FUNCTION_BLOCK FB_AlarmMAIN(*报警主功能块,请调用一次*)
VAR_INPUT
END_VAR
VAR_OUTPUT
	EventId:			DINT;(*报警号.有报警时会轮询输出有报警的id号*)
   	EventMessage:       WSTRING(255);(*报警信息.有报警时会轮询输出有报警的id信息*)
	EventAlive:			BOOL;(*当前有报警*)
	EventClass:			Alm_EventClass;(*当前的最大报警等级*)
  	NoStopAlarm:        BOOL;(*有小于7的报警,不停机报警*)
   	StopAlarm:          BOOL;(*有大于6的报警,停机报警*)
   	ShowlampOn:         BOOL;(*报警灯亮*)
   	FalshLamp:          BOOL;(*报警灯闪亮.有报警时该信号闪烁输出*)

	AutoRunOff:			BOOL;(*退出自动循环*)
	AlarmAction1:		BOOL;(*用户定义报警动作*)(*例如定义为黄灯亮,则有报警号有触发时,该输出信号为1*)
	AlarmAction2:		BOOL;(*用户定义报警动作*)
	AlarmAction3:		BOOL;(*用户定义报警动作*)
	AlarmAction4:		BOOL;(*用户定义报警动作*)
	AlarmAction5:		BOOL;(*用户定义报警动作*)
	AlarmAction6:		BOOL;(*用户定义报警动作*)
	AlarmAction7:		BOOL;(*用户定义报警动作*)
	AlarmAction8:		BOOL;(*用户定义报警动作*)
END_VAR
VAR
	nConut:                          DINT;
   	fbFreePluse:                     TON;
	m:                               DINT;
	Resul:                           DINT;
	n:                               DINT;
	R_TRIG_AlarmShow:        		 R_TRIG;
	R_TRIG_AlarmAlive:          	 R_TRIG;
	FB_FreePluse_AlarmShow: 		 TON;
	FB_FreePluse_AlarmAlive: 		 TON;
	F_TRIG_bHMIClearHistory: 		 F_TRIG;
	F_TRIG_EventAlive: 				 F_TRIG;
	InstLocalSystemTime:			 FB_LocalSystemTime;
END_VAR

(*Set Signal*)
 	EventAlive:=ShowlampOn:=AlarmAction1:=AlarmAction2:=AlarmAction3:=FALSE;
  	AlarmAction4:=AlarmAction5:=AlarmAction6:=AlarmAction7:=AlarmAction8:=FALSE;
	AutoRunOff :=	FALSE;(*退出自动循环*)
   	EventClass :=	0;

FOR nConut :=cnAlarmFirst TO cnAlarmLast DO
	    EventAlive :=	EventAlive OR AlarmActionArray[nConut].EventAlive;
	    ShowlampOn :=	ShowlampOn OR AlarmActionArray[nConut].ShowlampOn;
	    AlarmAction1:=	AlarmAction1 OR AlarmActionArray[nConut].AlarmAction1;
	    AlarmAction2:=	AlarmAction2 OR AlarmActionArray[nConut].AlarmAction2;
	    AlarmAction3:=	AlarmAction3 OR AlarmActionArray[nConut].AlarmAction3;
	    AlarmAction4:=	AlarmAction4 OR AlarmActionArray[nConut].AlarmAction4;
	    AlarmAction5:=	AlarmAction5 OR AlarmActionArray[nConut].AlarmAction5;
	    AlarmAction6:=	AlarmAction6 OR AlarmActionArray[nConut].AlarmAction6;
	    AlarmAction7:=	AlarmAction7 OR AlarmActionArray[nConut].AlarmAction7;
	    AlarmAction8:=	AlarmAction8 OR AlarmActionArray[nConut].AlarmAction8;
	    AutoRunOff :=	AutoRunOff 	OR AlarmActionArray[nConut].AutoRunOff;
	    EventClass  :=	MAX(EventClass,AlarmActionArray[nConut].EventClass);
END_FOR

(*Flash lamp*)
R_TRIG_AlarmShow(CLK:=ShowlampOn  );
IF ShowlampOn THEN              (****有报警时，先初始化时间输入为FALSE，灯亮，然后开始下步TON运行1S，闪灯状态变化
                                      优点：一有报警，就灯亮，避免有报警时过1S灯才亮*)
	IF R_TRIG_AlarmShow.Q THEN
		fbFreePluse(IN:=FALSE);
		FalshLamp:=TRUE;
	END_IF
	fbFreePluse(IN:=NOT fbFreePluse.Q,PT:=T#1S);
	IF fbFreePluse.Q THEN
		FalshLamp:=NOT FalshLamp;
	END_IF
ELSE
	FalshLamp:=FALSE;
END_IF



(*Action*)
AlarmAlive();
AlarmHMI();
AlarmShow();

(*Set Action*)
IF EventAlive THEN
     IF EventClass>6 THEN
         StopAlarm:=TRUE;
         NoStopAlarm:=FALSE;
     ELSE
         StopAlarm:=FALSE;
         NoStopAlarm:=TRUE;
    END_IF
ELSE
    StopAlarm:=FALSE;
    NoStopAlarm:=FALSE;
    EventId:=0;
    EventMessage:="";
    Alm_iHMIAlarmID:=0;
END_IF

	//获取系统时间
	InstLocalSystemTime(
		sNetID		:= '',
		bEnable		:= TRUE,
		dwCycle		:= 1,
		systemTime	=> tActSystemTime,
		);

ACTION AlarmAlive:
(*总报警数有n个，用其中有报警的[2],[4]赋值给激活报警m[1],[2],m自加1，然后循环比较m-20,把信息格式化*)
(*-----------------------------------当前报警列表显示-----------------------------*)
R_TRIG_AlarmAlive(CLK:=EventAlive);
IF EventAlive THEN
	IF R_TRIG_AlarmAlive.Q THEN
   	 	FB_FreePluse_AlarmAlive(In:=FALSE);
	END_IF
    FB_FreePluse_AlarmAlive(In:= NOT FB_FreePluse_AlarmAlive.Q,PT:=T#1S );
    IF FB_FreePluse_AlarmAlive.Q OR R_TRIG_AlarmAlive.Q THEN
         n:=cnAlarmFirst;
         m:=cnAlmActiveFirst;
          FOR n:=cnAlarmFirst TO cnAlarmLast DO     (*把所有报警赋值到当前激活报警数组*)
               IF AlarmActionArray[n].EventAlive THEN
                    AlarmActiveArray[m].EventId       :=AlarmActionArray[n].EventId;
                   	AlarmActiveArray[m].EventMessage  :=AlarmActionArray[n].EventMessage;						
                    AlarmActiveArray[m].EventTime     :=AlarmActionArray[n].EventTime;
                  	m:=m+1;
                    IF m>cnAlmActiveLast THEN
                       n:=32766;  (*exit FOR*)
                    END_IF
               END_IF
         END_FOR
         IF m<cnAlmActiveLast THEN
               FOR n:=m TO cnAlmActiveLast DO
                   AlarmActiveArray[n].EventId:=0;
                 	AlarmActiveArray[n].EventMessage:="";
                   	AlarmActiveArray[n].EventTime:=DT#2000-01-01-00:00;
             END_FOR
          END_IF
    END_IF
END_IF
(*当报警消失时,把显示列表内容清空*)
F_TRIG_EventAlive(CLK:=EventAlive );
IF F_TRIG_EventAlive.Q THEN
	FOR n:=cnAlmActiveFirst TO cnAlmActiveLast DO 
		AlarmActiveArray[n].EventId:=0;
		AlarmActiveArray[n].EventMessage:="";
		AlarmActiveArray[n].EventTime:=DT#2016-01-01-00:00;
	END_FOR
END_IF
END_ACTION

ACTION AlarmHMI:


(*``````````````````````````````````````````清除历史报警`````````````````````````````````````*)
F_TRIG_bHMIClearHistory(CLK:=Alm_bHMIClearHistory  );
IF F_TRIG_bHMIClearHistory.Q THEN
       FOR n:=cnAlmHistoryFirst TO cnAlmHistoryLast DO
             AlarmHistoryArray[n].EventId:=0;
             AlarmHistoryArray[n].EventMessage:="";
             AlarmHistoryArray[n].EventTime:=DT#2016-01-01-00:00;
        END_FOR
        Alm_HistoryAlarmNum:=0;
END_IF
END_ACTION

ACTION AlarmShow:

(*-------------------------------跑马灯显示报警---------------------------------*)
FB_FreePluse_AlarmShow(IN:=NOT FB_FreePluse_AlarmShow.Q,PT:=T#1S );
IF FB_FreePluse_AlarmShow.Q OR R_TRIG_AlarmAlive.Q THEN
      n:=EventId;
      	FOR m:=n+1 TO cnAlarmLast DO
            IF AlarmActionArray[m].EventAlive THEN
                   n:=m;
                   m:=cnAlarmLast+10;
             END_IF;
      	END_FOR;
    	IF n<>EventId THEN
        	Resul:=n;     
   		ELSE
          	FOR m:=cnAlarmFirst TO cnAlarmLast DO
             	IF AlarmActionArray[m].EventAlive THEN
                 	n:=m;
                 	m:=cnAlarmLast+10;
              	END_IF;
          	END_FOR;
          	Resul:=n;
      	END_IF
END_IF

Alm_iHMIAlarmID:=EventId:=Resul;
IF EventId<=cnAlarmLast AND EventId>= cnAlarmFirst THEN
	gwsActEventMsg:=EventMessage:=AlarmActionArray[EventId].EventMessage;
ELSE
	gwsActEventMsg:=EventMessage:="";	
END_IF
END_ACTION

END_FUNCTION_BLOCK

(* stored: Version 1.1.0.1, ProductVersion 3.1.4024.11
   POU FB_AlarmMain: Id {9dd3cfd5-45be-4f5b-9dd0-b9e05b59e1ce}, SpecialFunc None
   Action AlarmAlive: Id {07741066-2278-4707-a6ab-a8f3d50eecf5}
   Action AlarmHMI: Id {b8948498-7df0-420b-b573-3d450810b4de}
   Action AlarmShow: Id {b4465823-47e6-427a-9db5-86c5c2930f72} *)
